Universal Robots PolyScope program: Assembly_Vision.urp

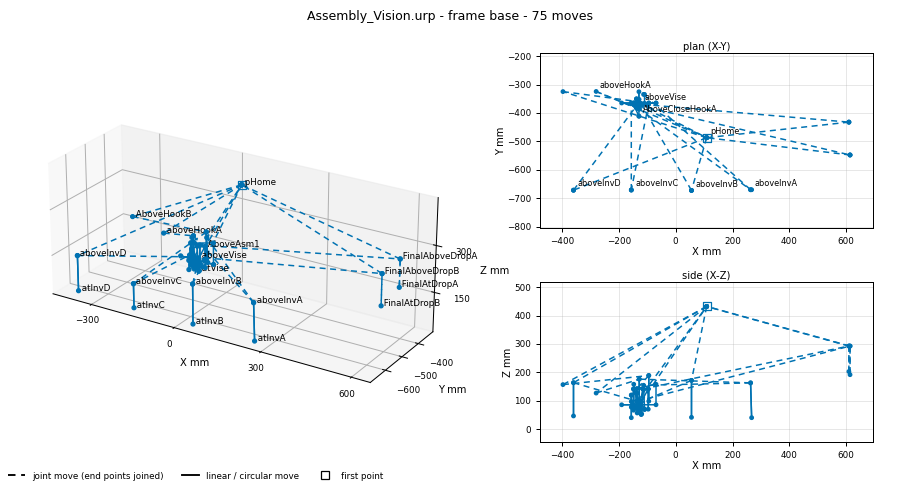
[picture p0: tool path of Assembly_Vision.urp in frame base, 75 of 75 moves have a stored position in this frame; points joined in program order, loops and branches not executed]
Program Assembly_Vision (installation=admin directory=/programs/THU_530PM/Final createdIn=3.15.8.106339 lastSavedIn=3.15.8.106339 robotSerialNumber=2015350926)
Calibrated DH parameters: a=[0, -0.425, -0.39225, 0, 0, 0]; d=[0.089159, 0, 0, 0.10915, 0.09465, 0.0823]; alpha=[1.570796, 0, 0, 1.570796, -1.570796, 0]; deltaTheta=[0, 0, 0, 0, 0, 0]
BeforeStart
  visionResult := 0
Robot Program (runOnlyOnce=true)
  SuppressedNode
    Script file /programs/THU_530PM/vision_pc_modbus.script
      | pc_ip = "10.241.34.37"
      | pc_port = 30002
      | 
      | connection = socket_open(pc_ip, pc_port, "vision_socket")
      | 
      | if (connection):
      |     socket_send_string("run_vision", "vision_socket")
      |     socket_close("vision_socket")
      | end
      | 
      | timeout = 15.0
      | elapsed =0.0
      | visionResult = 0
      | while visionResult == 0 and elapsed < timeout:
      |          sync()
      |          sleep(0.2)
      |          elapsed = elapsed + 0.2
      |          visionResult = modbus_get_signal_status ("vision_result")
      |          sync()
      | end
  Set DigitalOutput pin=digital_out[0]; digitalValue=0
  Set DigitalOutput pin=digital_out[1]; digitalValue=0
  If vision_result == 1 (checkContinuously=true)
    MoveJ speed 60 deg/s, acceleration 80 deg/s^2 (useActiveTCP=true)
      Waypoint pHome: TCP in base x=109.124 y=-486.883 z=431.849 mm, rx=0 ry=3.1416 rz=-0.0001 rad; joints [89.997, -90.004, 90.007, -90.008, -90, -0.002] deg
      Call _adminLinearIndex3
      Waypoint aboveInvB: TCP in base x=55.763 y=-672.337 z=171.801 mm, rx=0 ry=-3.1415 rz=-0.0001 rad; joints [85.431, -57.317, 86.752, -119.432, -90.004, -4.568] deg
    MoveL speed 250 mm/s, acceleration 1200 mm/s^2 (useActiveTCP=true) feature=Base
      Waypoint atInvB: TCP in base x=55.728 y=-672.308 z=41.705 mm, rx=-0.0002 ry=-3.1416 rz=-0.0003 rad; joints [85.428, -46.761, 91.224, -134.451, -90.002, -4.564] deg
      Set DigitalOutput pin=digital_out[0]; digitalValue=1
      Wait Sleep waitTime=1
      Waypoint aboveInvB: TCP in base x=55.763 y=-672.337 z=171.801 mm, rx=0 ry=-3.1415 rz=-0.0001 rad; joints [85.431, -57.317, 86.752, -119.432, -90.004, -4.568] deg
    MoveJ speed 60 deg/s, acceleration 80 deg/s^2 (useActiveTCP=true)
      Waypoint aboveVise: TCP in base x=-121.202 y=-368.6 z=95.842 mm, rx=0.0001 ry=-3.1413 rz=0.0004 rad; joints [55.461, -80.954, 138.438, -147.503, -90.004, -34.542] deg
    MoveL speed 250 mm/s, acceleration 1200 mm/s^2 (useActiveTCP=true) feature=Base
      Waypoint atVise: TCP in base x=-121.189 y=-368.616 z=51.473 mm, rx=0.0001 ry=-3.1414 rz=0.0005 rad; joints [55.463, -72.836, 139.996, -157.18, -90, -34.542] deg
      Set DigitalOutput pin=digital_out[0]; digitalValue=0
      Wait Sleep waitTime=1
      Waypoint aboveVise: TCP in base x=-121.202 y=-368.6 z=95.842 mm, rx=0.0001 ry=-3.1413 rz=0.0004 rad; joints [55.461, -80.954, 138.438, -147.503, -90.004, -34.542] deg
      Set DigitalOutput pin=digital_out[1]; digitalValue=1
    MoveJ speed 60 deg/s, acceleration 80 deg/s^2 (useActiveTCP=true)
      Waypoint pHome: TCP in base x=109.124 y=-486.883 z=431.849 mm, rx=0 ry=3.1416 rz=-0.0001 rad; joints [89.997, -90.004, 90.007, -90.008, -90, -0.002] deg
      Call _adminLinearIndex4
      Waypoint aboveHookA: TCP in base x=-279.674 y=-324.274 z=127.127 mm, rx=-2.2265 ry=2.2163 rz=-0.0001 rad; joints [34.456, -81.042, 130.829, -139.785, -89.997, -145.808] deg
    Call hookA_manager
    Call _adminLinearIndex3
    MoveJ speed 60 deg/s, acceleration 80 deg/s^2 (useActiveTCP=true)
      Waypoint aboveHookSlotA: TCP in base x=-128.133 y=-385.976 z=176.146 mm, rx=2.2264 ry=-2.2164 rz=0.0002 rad; joints [56.066, -90.044, 130.731, -130.689, -89.993, -124.193] deg
    MoveL speed 250 mm/s, acceleration 1200 mm/s^2 (useActiveTCP=true) feature=Base
      Waypoint atHookSlotA: TCP in base x=-128.351 y=-385.973 z=79.149 mm, rx=2.2265 ry=-2.2163 rz=0.0001 rad; joints [56.039, -76.105, 136.275, -150.175, -89.996, -124.224] deg
      Set DigitalOutput pin=digital_out[0]; digitalValue=0
      Wait Sleep waitTime=1
      Waypoint aboveHookSlotA: TCP in base x=-128.133 y=-385.976 z=176.146 mm, rx=2.2264 ry=-2.2164 rz=0.0002 rad; joints [56.066, -90.044, 130.731, -130.689, -89.993, -124.193] deg
    MoveJ speed 60 deg/s, acceleration 80 deg/s^2 (useActiveTCP=true)
      Waypoint aboveInvA: TCP in base x=263.578 y=-669.948 z=162.997 mm, rx=-0.0006 ry=-3.1415 rz=0.0003 rad; joints [102.757, -51.244, 77.791, -116.557, -90.006, 12.777] deg
    MoveL speed 250 mm/s, acceleration 1200 mm/s^2 (useActiveTCP=true) feature=Base
      Waypoint atInvA: TCP in base x=267.326 y=-669.929 z=40.528 mm, rx=-0.0004 ry=-3.1415 rz=0.0001 rad; joints [103.051, -41.912, 81.55, -129.639, -90.006, 13.065] deg
      Set DigitalOutput pin=digital_out[0]; digitalValue=1
      Wait Sleep waitTime=1
      Waypoint aboveInvA: TCP in base x=263.578 y=-669.948 z=162.997 mm, rx=-0.0006 ry=-3.1415 rz=0.0003 rad; joints [102.757, -51.244, 77.791, -116.557, -90.006, 12.777] deg
    MoveJ speed 60 deg/s, acceleration 80 deg/s^2 (useActiveTCP=true)
      Waypoint lidAPosAbove: TCP in base x=-112.743 y=-334.579 z=154.61 mm, rx=-0.0001 ry=-3.1414 rz=0.0003 rad; joints [53.37, -95.136, 139.767, -134.646, -90.003, -36.628] deg
    MoveL speed 50 mm/s, acceleration 100 mm/s^2 (useActiveTCP=true) feature=Base
      Waypoint lidAPos1: TCP in base x=-109.493 y=-334.537 z=71.015 mm, rx=0.0001 ry=-3.1414 rz=0.0003 rad; joints [53.813, -80.191, 144.9, -154.725, -90.003, -36.19] deg
      Waypoint lidAPos2: TCP in base x=-109.457 y=-365.942 z=69.152 mm, rx=0.0001 ry=-3.1414 rz=0.0003 rad; joints [56.743, -76.778, 140.419, -153.657, -90.001, -33.261] deg
      Set DigitalOutput pin=digital_out[0]; digitalValue=0
      Waypoint aboveVise: TCP in base x=-121.202 y=-368.6 z=95.842 mm, rx=0.0001 ry=-3.1413 rz=0.0004 rad; joints [55.461, -80.954, 138.438, -147.503, -90.004, -34.542] deg
      Set DigitalOutput pin=digital_out[0]; digitalValue=1
    MoveL speed 50 mm/s, acceleration 100 mm/s^2 (useActiveTCP=true) feature=Base
      Waypoint AboveAsm1: TCP in base x=-96.386 y=-369.771 z=141.514 mm, rx=0.0006 ry=-3.1414 rz=0.0004 rad; joints [58.794, -88.956, 136.696, -137.757, -90.003, -31.228] deg
      Waypoint AtAsm1: TCP in base x=-96.377 y=-369.785 z=70.442 mm, rx=-0.0007 ry=-3.1415 rz=0.0003 rad; joints [58.796, -77.006, 140.348, -153.355, -90.001, -31.179] deg
      Waypoint AboveAsm1: TCP in base x=-96.386 y=-369.771 z=141.514 mm, rx=0.0006 ry=-3.1414 rz=0.0004 rad; joints [58.794, -88.956, 136.696, -137.757, -90.003, -31.228] deg
      Waypoint AboveAsm2: TCP in base x=-148.343 y=-369.731 z=141.52 mm, rx=0.0002 ry=-3.1414 rz=0.0003 rad; joints [52.237, -86.763, 134.369, -137.621, -90.002, -37.771] deg
      Waypoint AtAsm2: TCP in base x=-148.301 y=-369.721 z=66.82 mm, rx=0.0003 ry=-3.1414 rz=0.0003 rad; joints [52.241, -74.772, 137.98, -153.224, -90.002, -37.77] deg
      Waypoint AboveAsm2: TCP in base x=-148.343 y=-369.731 z=141.52 mm, rx=0.0002 ry=-3.1414 rz=0.0003 rad; joints [52.237, -86.763, 134.369, -137.621, -90.002, -37.771] deg
      Waypoint AboveCloseHookA: TCP in base x=-129.172 y=-411.198 z=102.984 mm, rx=0.0003 ry=-3.1413 rz=0.0004 rad; joints [57.892, -77.309, 131.606, -144.32, -90.006, -32.118] deg
      Waypoint AtCloseHookA: TCP in base x=-129.164 y=-411.142 z=71.94 mm, rx=0.0002 ry=-3.1413 rz=0.0002 rad; joints [57.89, -72.563, 132.773, -150.226, -90.008, -32.118] deg
      Waypoint CloseHookA_1: TCP in base x=-129.177 y=-325.121 z=71.959 mm, rx=0.0001 ry=-3.1414 rz=0.0003 rad; joints [50.153, -80.619, 145.189, -154.585, -90.005, -39.85] deg
      Waypoint CloseHookA_2: TCP in base x=-129.145 y=-352.362 z=71.928 mm, rx=0.0002 ry=-3.1413 rz=0.0002 rad; joints [52.965, -77.974, 141.34, -153.381, -90.008, -37.043] deg
      Waypoint PressHookA: TCP in base x=-129.177 y=-352.405 z=70.909 mm, rx=0.0003 ry=-3.1413 rz=0.0002 rad; joints [52.965, -77.772, 141.368, -153.611, -90.008, -37.045] deg
      Waypoint AbovePickA: TCP in base x=-115.344 y=-369.772 z=141.51 mm, rx=0 ry=-3.1413 rz=0.0002 rad; joints [56.31, -88.241, 135.951, -137.724, -90.008, -33.691] deg
      Set DigitalOutput pin=digital_out[0]; digitalValue=0
      Waypoint AtPickA: TCP in base x=-119.449 y=-367.489 z=53.843 mm, rx=0 ry=-3.1414 rz=0.0002 rad; joints [55.588, -73.434, 140.184, -156.764, -90.007, -34.411] deg
      Set DigitalOutput pin=digital_out[1]; digitalValue=0
      Wait Sleep waitTime=0.5
      Set DigitalOutput pin=digital_out[0]; digitalValue=1
      Wait Sleep waitTime=1
      Waypoint AbovePickA: TCP in base x=-115.344 y=-369.772 z=141.51 mm, rx=0 ry=-3.1413 rz=0.0002 rad; joints [56.31, -88.241, 135.951, -137.724, -90.008, -33.691] deg
    MoveJ speed 60 deg/s, acceleration 80 deg/s^2 (useActiveTCP=true)
      Waypoint FinalAboveDropA: TCP in base x=609.432 y=-432.167 z=292.569 mm, rx=-0.0003 ry=3.1416 rz=-0.0003 rad; joints [136.258, -52.983, 60.844, -97.87, -90.008, 46.247] deg
      Waypoint FinalAtDropA: TCP in base x=609.419 y=-432.13 z=202.922 mm, rx=0.0004 ry=-3.1415 rz=0.0001 rad; joints [136.26, -49.867, 69.047, -109.179, -90.007, 46.245] deg
      Set DigitalOutput pin=digital_out[0]; digitalValue=0
      Wait Sleep waitTime=1
      Waypoint FinalAboveDropA: TCP in base x=609.432 y=-432.167 z=292.569 mm, rx=-0.0003 ry=3.1416 rz=-0.0003 rad; joints [136.258, -52.983, 60.844, -97.87, -90.008, 46.247] deg
    MoveJ speed 60 deg/s, acceleration 80 deg/s^2 (useActiveTCP=true)
      Waypoint pHome: TCP in base x=109.124 y=-486.883 z=431.849 mm, rx=0 ry=3.1416 rz=-0.0001 rad; joints [89.997, -90.004, 90.007, -90.008, -90, -0.002] deg
  ElseIf vision_result == 2 (checkContinuously=true)
    MoveJ speed 60 deg/s, acceleration 80 deg/s^2 (useActiveTCP=true)
      Waypoint pHome: TCP in base x=109.124 y=-486.883 z=431.849 mm, rx=0 ry=3.1416 rz=-0.0001 rad; joints [89.997, -90.004, 90.007, -90.008, -90, -0.002] deg
      Call _adminLinearIndex3
      Waypoint aboveInvD: TCP in base x=-359.322 y=-671.519 z=163.591 mm, rx=0 ry=3.1415 rz=0 rad; joints [53.609, -45.864, 68.075, -112.208, -89.994, -36.391] deg
    MoveL speed 250 mm/s, acceleration 1200 mm/s^2 (useActiveTCP=true) feature=Base
      Waypoint atInvD: TCP in base x=-359.329 y=-671.527 z=46.641 mm, rx=0 ry=-3.1416 rz=0.0003 rad; joints [53.609, -37.915, 72.276, -124.37, -89.994, -36.391] deg
      Set DigitalOutput pin=digital_out[0]; digitalValue=1
      Wait Sleep waitTime=1
      Waypoint aboveInvD: TCP in base x=-359.322 y=-671.519 z=163.591 mm, rx=0 ry=3.1415 rz=0 rad; joints [53.609, -45.864, 68.075, -112.208, -89.994, -36.391] deg
    MoveJ speed 60 deg/s, acceleration 80 deg/s^2 (useActiveTCP=true)
      Waypoint AboveVise_B: TCP in base x=-135.429 y=-371.917 z=98.365 mm, rx=0.0001 ry=-3.1413 rz=0.0002 rad; joints [53.986, -80.494, 137.151, -146.672, -90.008, -36.018] deg
    MoveL speed 250 mm/s, acceleration 1200 mm/s^2 (useActiveTCP=true) feature=Base
      Waypoint AtVise_B: TCP in base x=-135.424 y=-371.942 z=57.173 mm, rx=0.0001 ry=-3.1413 rz=0.0003 rad; joints [53.988, -73.24, 138.645, -155.425, -90.008, -36.017] deg
      Set DigitalOutput pin=digital_out[0]; digitalValue=0
      Wait Sleep waitTime=1
      Waypoint AboveVise_B: TCP in base x=-135.429 y=-371.917 z=98.365 mm, rx=0.0001 ry=-3.1413 rz=0.0002 rad; joints [53.986, -80.494, 137.151, -146.672, -90.008, -36.018] deg
      Set DigitalOutput pin=digital_out[1]; digitalValue=1
    MoveJ speed 60 deg/s, acceleration 80 deg/s^2 (useActiveTCP=true)
      Waypoint pHome: TCP in base x=109.124 y=-486.883 z=431.849 mm, rx=0 ry=3.1416 rz=-0.0001 rad; joints [89.997, -90.004, 90.007, -90.008, -90, -0.002] deg
      Call _adminLinearIndex4
      Waypoint AboveHookB: TCP in base x=-396.369 y=-324.75 z=156.893 mm, rx=-2.2267 ry=2.2162 rz=0 rad; joints [27.029, -74.692, 116.186, -131.493, -90, -153.241] deg
    Folder HookBManager
      above_HookB := p[-0.39636, -0.32475, 0.15692, 2.226, -2.216, 0.000]
      offset_x := hook_indexB * 0.047
      above_pose_B := pose_add(above_HookB, p[0.0, -offset_x, 0.0, 0.0, 0.0, 0.0])
      at_pose_B := pose_add(above_pose_B, p[0.0, 0.0, -0.10503, 0.0, 0.0, 0.0])
      Script: movel (get_inverse_kin(above_pose_B))
      Script: movel (get_inverse_kin(at_pose_B))
      Set DigitalOutput pin=digital_out[0]; digitalValue=1
      Wait Sleep waitTime=1
      Script: movel (get_inverse_kin(above_pose_B), a = 0.5, v = 0.1)
      Script: movej (get_inverse_kin(above_HookB))
      hook_indexB := hook_indexB + 1
      If hook_index ≥ num_hooks
        hook_indexB := 0
        Popup Message (haltProgram=false message=All Hook_B's were used! Reload Fixture inputType=Text)
    Call _adminLinearIndex3
    MoveJ speed 60 deg/s, acceleration 80 deg/s^2 (useActiveTCP=true)
      Waypoint AboveHookSlotB: TCP in base x=-94.499 y=-365.185 z=188.889 mm, rx=-3.1415 ry=-0.0009 rz=-0.0001 rad; joints [58.672, -95.839, 133.703, -127.859, -89.999, -211.362] deg
    MoveL speed 250 mm/s, acceleration 1200 mm/s^2 (useActiveTCP=true) feature=Base
      Waypoint AtHookSlotB: TCP in base x=-94.512 y=-365.178 z=98.575 mm, rx=-3.1414 ry=-0.0024 rz=-0.0001 rad; joints [58.671, -82.686, 139.912, -147.217, -90.003, -211.418] deg
      Set DigitalOutput pin=digital_out[0]; digitalValue=0
      Wait Sleep waitTime=1
      Waypoint AboveHookSlotB: TCP in base x=-94.499 y=-365.185 z=188.889 mm, rx=-3.1415 ry=-0.0009 rz=-0.0001 rad; joints [58.672, -95.839, 133.703, -127.859, -89.999, -211.362] deg
    MoveJ speed 60 deg/s, acceleration 80 deg/s^2 (useActiveTCP=true)
      Waypoint aboveInvC: TCP in base x=-156.001 y=-670.82 z=119.963 mm, rx=-0.0001 ry=-3.1416 rz=0.0002 rad; joints [67.789, -51.979, 86.398, -124.427, -89.997, -22.208] deg
    MoveL speed 250 mm/s, acceleration 1200 mm/s^2 (useActiveTCP=true) feature=Base
      Waypoint atInvC: TCP in base x=-155.967 y=-670.825 z=40.553 mm, rx=0 ry=-3.1416 rz=0.0003 rad; joints [67.792, -45.263, 88.405, -133.151, -89.997, -22.21] deg
      Set DigitalOutput pin=digital_out[0]; digitalValue=1
      Wait Sleep waitTime=1
      Waypoint aboveInvC: TCP in base x=-156.001 y=-670.82 z=119.963 mm, rx=-0.0001 ry=-3.1416 rz=0.0002 rad; joints [67.789, -51.979, 86.398, -124.427, -89.997, -22.208] deg
    MoveJ speed 60 deg/s, acceleration 80 deg/s^2 (useActiveTCP=true)
      Waypoint lidBPosAbove: TCP in base x=-156 y=-365.975 z=97.411 mm, rx=0.0001 ry=3.1415 rz=0 rad; joints [50.989, -80.11, 136.885, -146.774, -89.996, -39.007] deg
    MoveL speed 50 mm/s, acceleration 100 mm/s^2 (useActiveTCP=true) feature=Base
      Waypoint LidBPos1: TCP in base x=-155.989 y=-364.37 z=77.485 mm, rx=0.0001 ry=3.1416 rz=-0.0001 rad; joints [50.838, -76.868, 137.926, -151.062, -89.996, -39.16] deg
      Waypoint LidBPos2: TCP in base x=-128.709 y=-364.962 z=74.096 mm, rx=0.0002 ry=3.1415 rz=-0.0002 rad; joints [54.19, -77.204, 139.477, -152.275, -89.992, -35.805] deg
      Set DigitalOutput pin=digital_out[0]; digitalValue=0
      Wait Sleep waitTime=1
      Waypoint AboveVise_B: TCP in base x=-135.429 y=-371.917 z=98.365 mm, rx=0.0001 ry=-3.1413 rz=0.0002 rad; joints [53.986, -80.494, 137.151, -146.672, -90.008, -36.018] deg
      Set DigitalOutput pin=digital_out[0]; digitalValue=1
    MoveL speed 50 mm/s, acceleration 100 mm/s^2 (useActiveTCP=true) feature=Base
      Waypoint AboveAsmB1: TCP in base x=-137.641 y=-381.922 z=127.91 mm, rx=0 ry=3.1415 rz=-0.0001 rad; joints [54.583, -83.859, 134.094, -140.237, -89.993, -35.416] deg
      Waypoint AtAsmB1: TCP in base x=-137.623 y=-381.875 z=75.465 mm, rx=0 ry=3.1415 rz=-0.0002 rad; joints [54.581, -75.561, 136.533, -150.975, -89.992, -35.417] deg
      Waypoint AboveAsmB1: TCP in base x=-137.641 y=-381.922 z=127.91 mm, rx=0 ry=3.1415 rz=-0.0001 rad; joints [54.583, -83.859, 134.094, -140.237, -89.993, -35.416] deg
      Waypoint AboveAsmB2: TCP in base x=-137.641 y=-350.614 z=126.29 mm, rx=0.0001 ry=3.1415 rz=-0.0003 rad; joints [51.72, -87.389, 138.459, -141.076, -89.991, -38.277] deg
      Waypoint AtAsmB2: TCP in base x=-137.719 y=-350.629 z=73.666 mm, rx=-0.0003 ry=-3.1408 rz=0.002 rad; joints [51.711, -78.151, 141.082, -153.019, -89.991, -38.28] deg
      Waypoint AboveAsmB2: TCP in base x=-137.641 y=-350.614 z=126.29 mm, rx=0.0001 ry=3.1415 rz=-0.0003 rad; joints [51.72, -87.389, 138.459, -141.076, -89.991, -38.277] deg
      Waypoint ToCloseHook: TCP in base x=-136.305 y=-368.201 z=143.224 mm, rx=0.0001 ry=-3.1414 rz=0.0003 rad; joints [53.546, -87.77, 135.085, -137.332, -90.004, -36.459] deg
      Waypoint AboveHookClose: TCP in base x=-69.041 y=-364.899 z=158.13 mm, rx=0.0002 ry=3.1415 rz=0.0001 rad; joints [62.193, -92.852, 136.996, -134.137, -89.996, -27.8] deg
      Waypoint AtHookClose: TCP in base x=-69.072 y=-364.875 z=86.018 mm, rx=0.0001 ry=3.1414 rz=0.0002 rad; joints [62.186, -81.079, 141.368, -150.277, -89.994, -27.809] deg
      Waypoint HookClose: TCP in base x=-189.861 y=-364.857 z=85.992 mm, rx=0.0002 ry=3.1415 rz=0.0003 rad; joints [47.12, -76.78, 135.319, -148.528, -90.003, -42.872] deg
      Waypoint CloseHookPos1: TCP in base x=-147.092 y=-364.909 z=86.076 mm, rx=0.0001 ry=3.1415 rz=-0.0001 rad; joints [51.938, -78.673, 138.04, -149.369, -89.994, -38.059] deg
      Waypoint CloseHookPos2: TCP in base x=-147.049 y=-364.912 z=78.564 mm, rx=-0.0001 ry=3.1416 rz=0 rad; joints [51.944, -77.357, 138.333, -150.976, -89.998, -38.058] deg
    MoveL speed 250 mm/s, acceleration 1200 mm/s^2 (useActiveTCP=true) feature=Base
      Waypoint AboveVise: TCP in base x=-147.373 y=-364.918 z=158.17 mm, rx=0.0003 ry=3.1414 rz=0 rad; joints [51.905, -89.668, 133.91, -134.234, -89.993, -38.084] deg
      Set DigitalOutput pin=digital_out[0]; digitalValue=0
      Waypoint AtPickB: TCP in base x=-130.247 y=-364.91 z=59.515 mm, rx=0.0002 ry=3.1414 rz=0.0001 rad; joints [53.993, -74.434, 139.868, -155.425, -89.993, -35.998] deg
      Set DigitalOutput pin=digital_out[1]; digitalValue=0
      Wait Sleep waitTime=1
      Set DigitalOutput pin=digital_out[0]; digitalValue=1
      Wait Sleep waitTime=1
      Waypoint AboveVise_B: TCP in base x=-135.429 y=-371.917 z=98.365 mm, rx=0.0001 ry=-3.1413 rz=0.0002 rad; joints [53.986, -80.494, 137.151, -146.672, -90.008, -36.018] deg
    MoveJ speed 60 deg/s, acceleration 80 deg/s^2 (useActiveTCP=true)
      Waypoint FinalAboveDropB: TCP in base x=613.435 y=-547.672 z=292.561 mm, rx=0.0004 ry=-3.1416 rz=0.0002 rad; joints [130.615, -39.384, 37.044, -87.666, -90.006, 40.601] deg
      Waypoint FinalAtDropB: TCP in base x=613.407 y=-547.713 z=191.767 mm, rx=-0.0003 ry=3.1415 rz=-0.0004 rad; joints [130.611, -37.854, 49.012, -101.171, -90.005, 40.602] deg
      Set DigitalOutput pin=digital_out[0]; digitalValue=0
      Wait Sleep waitTime=1
      Waypoint FinalAboveDropB: TCP in base x=613.435 y=-547.672 z=292.561 mm, rx=0.0004 ry=-3.1416 rz=0.0002 rad; joints [130.615, -39.384, 37.044, -87.666, -90.006, 40.601] deg
    MoveJ speed 60 deg/s, acceleration 80 deg/s^2 (useActiveTCP=true)
      Waypoint pHome: TCP in base x=109.124 y=-486.883 z=431.849 mm, rx=0 ry=3.1416 rz=-0.0001 rad; joints [89.997, -90.004, 90.007, -90.008, -90, -0.002] deg
SubProgram -> hookA_manager
SubProgram -> _adminLinearIndex4
SubProgram -> _adminLinearIndex3
SubProgram _adminLinearIndex2 (keepSynchronizedWithDisk=false) programFile=/programs/me345_admin/_adminLinearIndex2.urp
  Folder Move_linear_slide_Index2
    var_1 := False
    Loop While (checkContinuously=false) expression=var_1≟ False
      var_1 := socket_open("10.241.34.44",4001)
    var_3 := 1
    Send := "s r0x24 21"
    Script: socket_send_string(Send)
    Script: socket_send_byte(13)
    Send_Reply := socket_read_string()
    Send := "s r0xca 51968"
    Script: socket_send_string(Send)
    Script: socket_send_byte(13)
    Send_Reply := socket_read_string()
    Send := "t 1"
    Script: socket_send_string(Send)
    Script: socket_send_byte(13)
    Send_Reply := socket_read_string()
    Loop While (checkContinuously=false) expression=var_3≠0
      Send := "g r0xA0"
      Script: socket_send_string(Send)
      Script: socket_send_byte(13)
      var_3 := socket_get_var("v")
      Wait Sleep waitTime=0.1
    Script: socket_close()
    Script: sync()
SubProgram _adminLinearIndex5 (keepSynchronizedWithDisk=false) programFile=/programs/me345_admin/_adminLinearIndex5.urp
  Folder Move_linear_slide_Index5
    var_1 := False
    Loop While (checkContinuously=false) expression=var_1≟ False
      var_1 := socket_open("10.241.34.44",4001)
    var_3 := 1
    Send := "s r0x24 21"
    Script: socket_send_string(Send)
    Script: socket_send_byte(13)
    Send_Reply := socket_read_string()
    Send := "s r0xca 190000"
    Script: socket_send_string(Send)
    Script: socket_send_byte(13)
    Send_Reply := socket_read_string()
    Send := "t 1"
    Script: socket_send_string(Send)
    Script: socket_send_byte(13)
    Send_Reply := socket_read_string()
    Loop While (checkContinuously=false) expression=var_3≠0
      Send := "g r0xA0"
      Script: socket_send_string(Send)
      Script: socket_send_byte(13)
      var_3 := socket_get_var("v")
      Wait Sleep waitTime=0.1
    Script: socket_close()
    Script: sync()
SubProgram _adminLinearIndex3 (keepSynchronizedWithDisk=false) programFile=/programs/me345_admin/_adminLinearIndex3.urp
  Folder Move_linear_slide_Index1
    var_1 := False
    Loop While (checkContinuously=false) expression=var_1≟ False
      var_1 := socket_open("10.241.34.44",4001)
    var_3 := 1
    Send := "s r0x24 21"
    Script: socket_send_string(Send)
    Script: socket_send_byte(13)
    Send_Reply := socket_read_string()
    Send := "s r0xca 103936"
    Script: socket_send_string(Send)
    Script: socket_send_byte(13)
    Send_Reply := socket_read_string()
    Send := "t 1"
    Script: socket_send_string(Send)
    Script: socket_send_byte(13)
    Send_Reply := socket_read_string()
    Loop While (checkContinuously=false) expression=var_3≠0
      Send := "g r0xA0"
      Script: socket_send_string(Send)
      Script: socket_send_byte(13)
      var_3 := socket_get_var("v")
      Wait Sleep waitTime=0.1
    Script: socket_close()
    Script: sync()
SubProgram _adminLinearIndex4 (keepSynchronizedWithDisk=false) programFile=/programs/me345_admin/_adminLinearIndex4.urp
  Folder Move_linear_slide_Index1
    var_1 := False
    Loop While (checkContinuously=false) expression=var_1≟ False
      var_1 := socket_open("10.241.34.44",4001)
    var_3 := 1
    Send := "s r0x24 21"
    Script: socket_send_string(Send)
    Script: socket_send_byte(13)
    Send_Reply := socket_read_string()
    Send := "s r0xca 155904"
    Script: socket_send_string(Send)
    Script: socket_send_byte(13)
    Send_Reply := socket_read_string()
    Send := "t 1"
    Script: socket_send_string(Send)
    Script: socket_send_byte(13)
    Send_Reply := socket_read_string()
    Loop While (checkContinuously=false) expression=var_3≠0
      Send := "g r0xA0"
      Script: socket_send_string(Send)
      Script: socket_send_byte(13)
      var_3 := socket_get_var("v")
      Wait Sleep waitTime=0.1
    Script: socket_close()
    Script: sync()
SubProgram hookA_manager (keepSynchronizedWithDisk=false) programFile=/programs/THU_530PM/hookA_manager.urp
  above_HookA := p[-0.27970, -0.32422, 0.12715, 2.226, -2.216, 0.000]
  offset_x := hook_index * 0.047
  above_pose_A := pose_add(above_HookA, p[0.0, -offset_x, 0.0, 0.0, 0.0, 0.0])
  at_pose_A := pose_add(above_pose_A, p[0.0, 0.0, -0.086, 0.0, 0.0, 0.0])
  Script: movel (get_inverse_kin(above_pose_A))
  Script: movel (get_inverse_kin(at_pose_A))
  Set DigitalOutput pin=digital_out[0]; digitalValue=1
  Wait Sleep waitTime=1
  Script: movel (get_inverse_kin(above_pose_A), a = 0.5, v = 0.1)
  Script: movej (get_inverse_kin(above_HookA))
  hook_index := hook_index + 1
  If hook_index ≥ num_hooks
    hook_index := 0
    Popup Message (haltProgram=false message=All Hook_A's were used! Reload Fixture inputType=Text)
